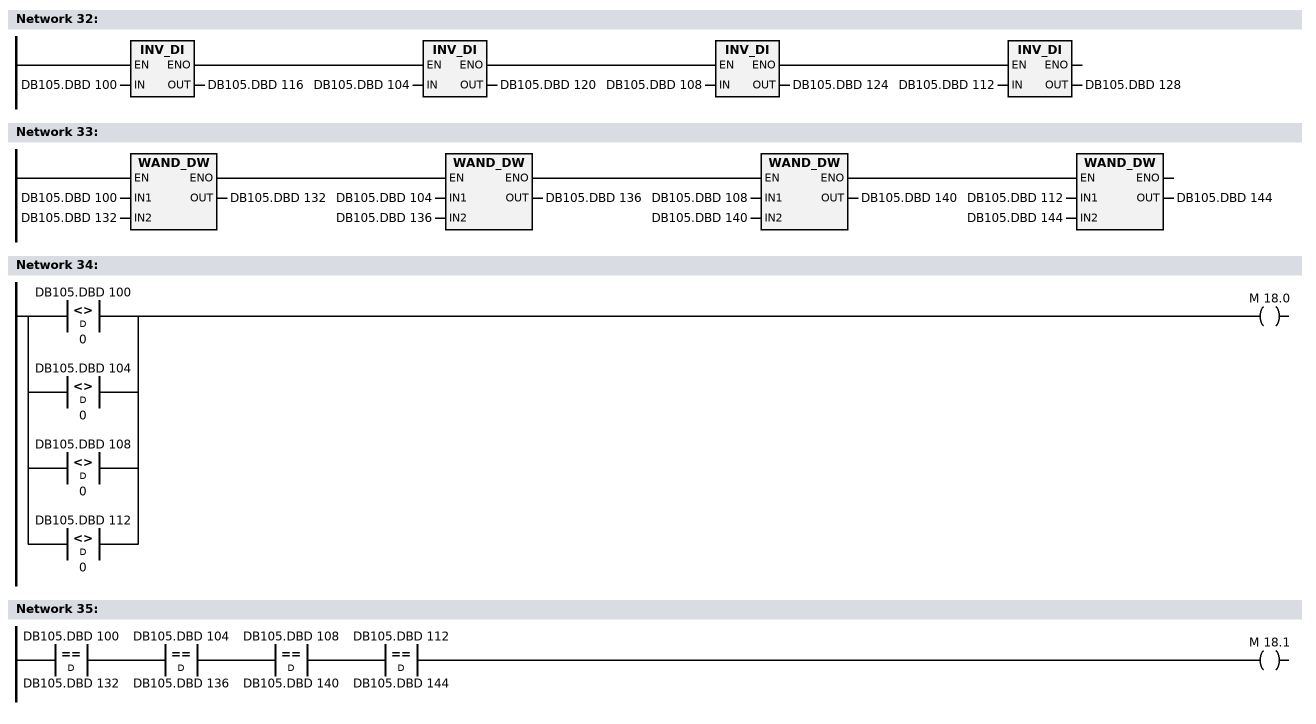
NETWORK
TITLE =
      A(;
      A(;
      A(;
      L     DB105.DBD 100;
      INVD;
      T     DB105.DBD 116;
      SET;
      SAVE;
      CLR;
      A     BR;
      );
      JNB   M001;
      L     DB105.DBD 104;
      INVD;
      T     DB105.DBD 120;
      SET;
      SAVE;
      CLR;
M001: A     BR;
      );
      JNB   M002;
      L     DB105.DBD 108;
      INVD;
      T     DB105.DBD 124;
      SET;
      SAVE;
      CLR;
M002: A     BR;
      );
      JNB   M003;
      L     DB105.DBD 112;
      INVD;
      T     DB105.DBD 128;
M003: NOP   0;
NETWORK
TITLE =
      A(;
      A(;
      A(;
      L     DB105.DBD 100;
      L     DB105.DBD 132;
      AD;
      T     DB105.DBD 132;
      SET;
      SAVE;
      CLR;
      A     BR;
      );
      JNB   M004;
      L     DB105.DBD 104;
      L     DB105.DBD 136;
      AD;
      T     DB105.DBD 136;
      SET;
      SAVE;
      CLR;
M004: A     BR;
      );
      JNB   M005;
      L     DB105.DBD 108;
      L     DB105.DBD 140;
      AD;
      T     DB105.DBD 140;
      SET;
      SAVE;
      CLR;
M005: A     BR;
      );
      JNB   M006;
      L     DB105.DBD 112;
      L     DB105.DBD 144;
      AD;
      T     DB105.DBD 144;
M006: NOP   0;
NETWORK
TITLE =
      O(;
      L     DB105.DBD 100;
      L     0;
      <>D;
      );
      O(;
      L     DB105.DBD 104;
      L     0;
      <>D;
      );
      O(;
      L     DB105.DBD 108;
      L     0;
      <>D;
      );
      O(;
      L     DB105.DBD 112;
      L     0;
      <>D;
      );
      =     M 18.0;
NETWORK
TITLE =
      A(;
      L     DB105.DBD 100;
      L     DB105.DBD 132;
      ==D;
      );
      A(;
      L     DB105.DBD 104;
      L     DB105.DBD 136;
      ==D;
      );
      A(;
      L     DB105.DBD 108;
      L     DB105.DBD 140;
      ==D;
      );
      A(;
      L     DB105.DBD 112;
      L     DB105.DBD 144;
      ==D;
      );
      =     M 18.1;
END_FUNCTION

FUNCTION FC 119 : VOID
VERSION : 0.1
BEGIN
// (block stored without names or comments; labels and parameter names are numbered)
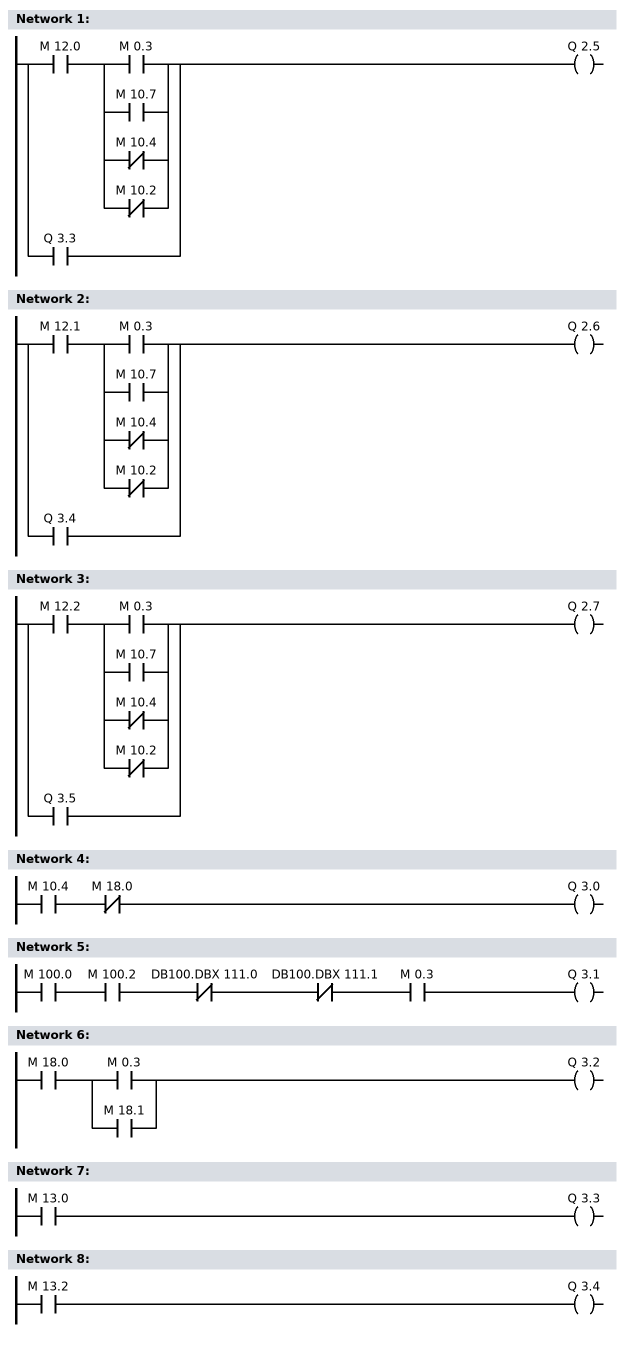
NETWORK
TITLE =
      A     M 12.0;
      A(;
      O     M 0.3;
      O     M 10.7;
      ON    M 10.4;
      ON    M 10.2;
      );
      O     Q 3.3;
      =     Q 2.5;
NETWORK
TITLE =
      A     M 12.1;
      A(;
      O     M 0.3;
      O     M 10.7;
      ON    M 10.4;
      ON    M 10.2;
      );
      O     Q 3.4;
      =     Q 2.6;
NETWORK
TITLE =
      A     M 12.2;
      A(;
      O     M 0.3;
      O     M 10.7;
      ON    M 10.4;
      ON    M 10.2;
      );
      O     Q 3.5;
      =     Q 2.7;
NETWORK
TITLE =
      A     M 10.4;
      AN    M 18.0;
      =     Q 3.0;
NETWORK
TITLE =
      A     M 100.0;
      A     M 100.2;
      AN    DB100.DBX 111.0;
      AN    DB100.DBX 111.1;
      A     M 0.3;
      =     Q 3.1;
NETWORK
TITLE =
      A     M 18.0;
      A(;
      O     M 0.3;
      O     M 18.1;
      );
      =     Q 3.2;
NETWORK
TITLE =
      A     M 13.0;
      =     Q 3.3;
NETWORK
TITLE =
      A     M 13.2;
      =     Q 3.4;
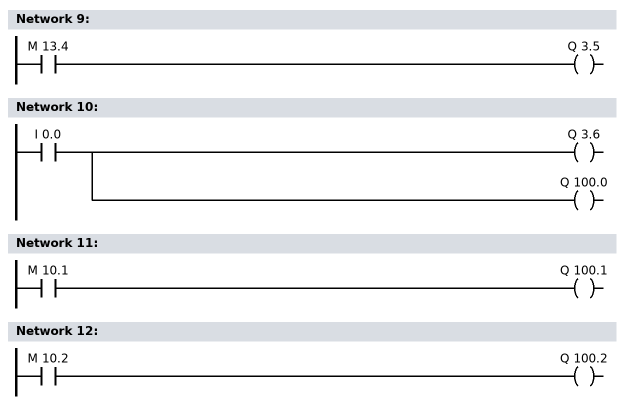
NETWORK
TITLE =
      A     M 13.4;
      =     Q 3.5;
NETWORK
TITLE =
      A     I 0.0;
      =     Q 3.6;
      =     Q 100.0;
NETWORK
TITLE =
      A     M 10.1;
      =     Q 100.1;
NETWORK
TITLE =
      A     M 10.2;
      =     Q 100.2;
END_FUNCTION

FUNCTION FC 140 : VOID
VERSION : 0.1
BEGIN
// (block stored without names or comments; labels and parameter names are numbered)
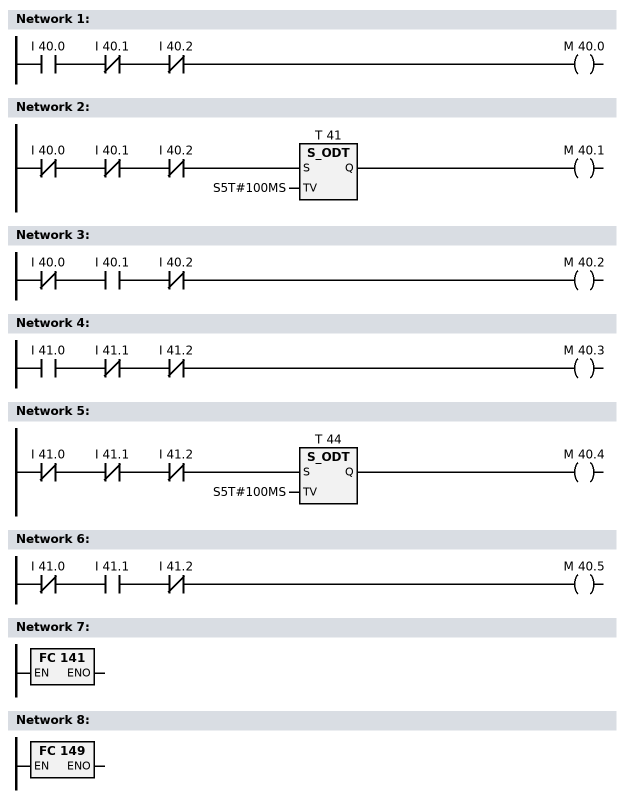
NETWORK
TITLE =
      A     I 40.0;
      AN    I 40.1;
      AN    I 40.2;
      =     M 40.0;
NETWORK
TITLE =
      AN    I 40.0;
      AN    I 40.1;
      AN    I 40.2;
      L     S5T#100MS;
      SD    T 41;
      NOP   0;
      NOP   0;
      NOP   0;
      A     T 41;
      =     M 40.1;
NETWORK
TITLE =
      AN    I 40.0;
      A     I 40.1;
      AN    I 40.2;
      =     M 40.2;
NETWORK
TITLE =
      A     I 41.0;
      AN    I 41.1;
      AN    I 41.2;
      =     M 40.3;
NETWORK
TITLE =
      AN    I 41.0;
      AN    I 41.1;
      AN    I 41.2;
      L     S5T#100MS;
      SD    T 44;
      NOP   0;
      NOP   0;
      NOP   0;
      A     T 44;
      =     M 40.4;
NETWORK
TITLE =
      AN    I 41.0;
      A     I 41.1;
      AN    I 41.2;
      =     M 40.5;
NETWORK
TITLE =
      CALL  FC 141;
      NOP   0;
NETWORK
TITLE =
      CALL  FC 149;
      NOP   0;
END_FUNCTION

FUNCTION FC 141 : VOID
VERSION : 0.1
BEGIN
// (block stored without names or comments; labels and parameter names are numbered)
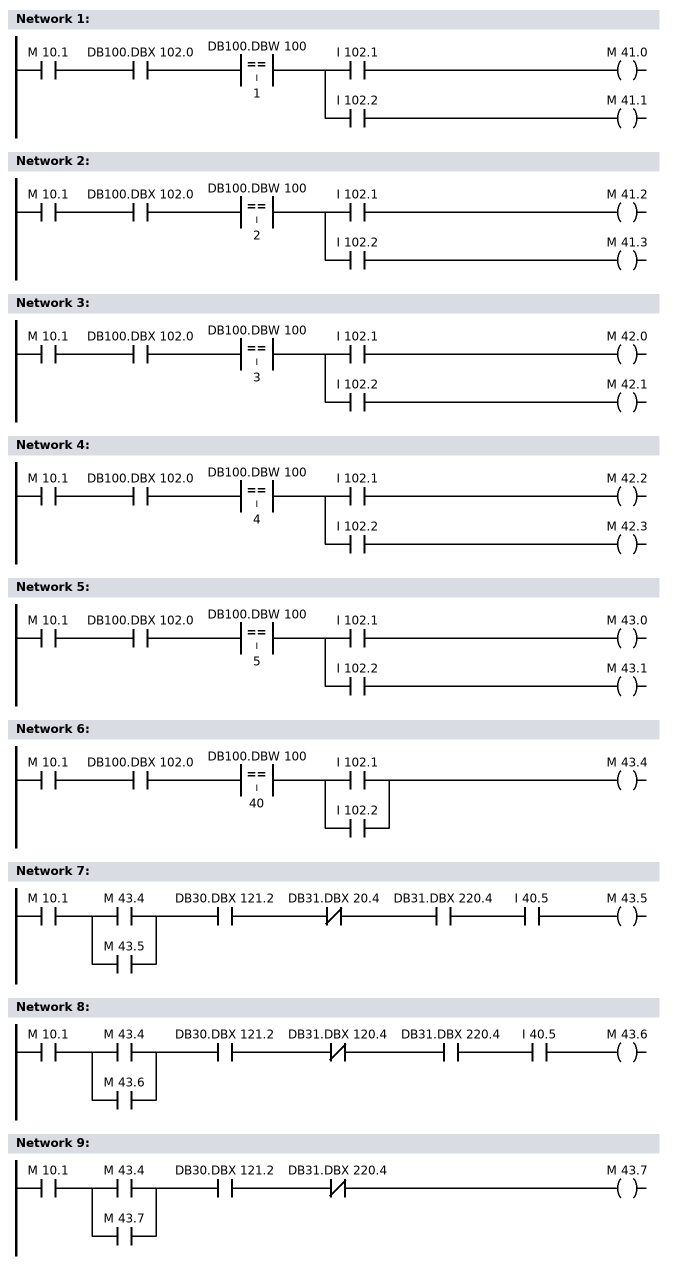
NETWORK
TITLE =
      A     M 10.1;
      A     DB100.DBX 102.0;
      A(;
      L     DB100.DBW 100;
      L     1;
      ==I;
      );
      =     L 0.0;
      A     L 0.0;
      A     I 102.1;
      =     M 41.0;
      A     L 0.0;
      A     I 102.2;
      =     M 41.1;
NETWORK
TITLE =
      A     M 10.1;
      A     DB100.DBX 102.0;
      A(;
      L     DB100.DBW 100;
      L     2;
      ==I;
      );
      =     L 0.0;
      A     L 0.0;
      A     I 102.1;
      =     M 41.2;
      A     L 0.0;
      A     I 102.2;
      =     M 41.3;
NETWORK
TITLE =
      A     M 10.1;
      A     DB100.DBX 102.0;
      A(;
      L     DB100.DBW 100;
      L     3;
      ==I;
      );
      =     L 0.0;
      A     L 0.0;
      A     I 102.1;
      =     M 42.0;
      A     L 0.0;
      A     I 102.2;
      =     M 42.1;
NETWORK
TITLE =
      A     M 10.1;
      A     DB100.DBX 102.0;
      A(;
      L     DB100.DBW 100;
      L     4;
      ==I;
      );
      =     L 0.0;
      A     L 0.0;
      A     I 102.1;
      =     M 42.2;
      A     L 0.0;
      A     I 102.2;
      =     M 42.3;
NETWORK
TITLE =
      A     M 10.1;
      A     DB100.DBX 102.0;
      A(;
      L     DB100.DBW 100;
      L     5;
      ==I;
      );
      =     L 0.0;
      A     L 0.0;
      A     I 102.1;
      =     M 43.0;
      A     L 0.0;
      A     I 102.2;
      =     M 43.1;
NETWORK
TITLE =
      A     M 10.1;
      A     DB100.DBX 102.0;
      A(;
      L     DB100.DBW 100;
      L     40;
      ==I;
      );
      A(;
      O     I 102.1;
      O     I 102.2;
      );
      =     M 43.4;
NETWORK
TITLE =
      A     M 10.1;
      A(;
      O     M 43.4;
      O     M 43.5;
      );
      A     DB30.DBX 121.2;
      AN    DB31.DBX 20.4;
      A     DB31.DBX 220.4;
      A     I 40.5;
      =     M 43.5;
NETWORK
TITLE =
      A     M 10.1;
      A(;
      O     M 43.4;
      O     M 43.6;
      );
      A     DB30.DBX 121.2;
      AN    DB31.DBX 120.4;
      A     DB31.DBX 220.4;
      A     I 40.5;
      =     M 43.6;
NETWORK
TITLE =
      A     M 10.1;
      A(;
      O     M 43.4;
      O     M 43.7;
      );
      A     DB30.DBX 121.2;
      AN    DB31.DBX 220.4;
      =     M 43.7;
END_FUNCTION

FUNCTION FC 142 : VOID
VERSION : 0.1
BEGIN
// (block stored without names or comments; labels and parameter names are numbered)
END_FUNCTION

FUNCTION FC 149 : VOID
VERSION : 0.1
BEGIN
// (block stored without names or comments; labels and parameter names are numbered)
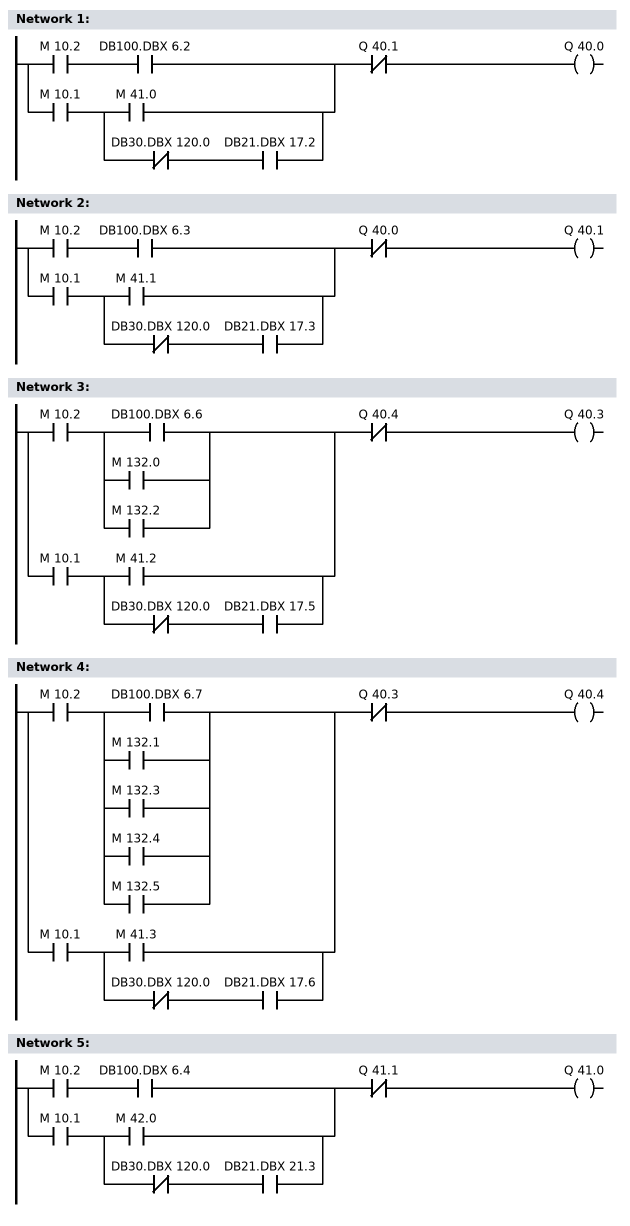
NETWORK
TITLE =
      A(;
      A     M 10.2;
      A     DB100.DBX 6.2;
      O;
      A     M 10.1;
      A(;
      O     M 41.0;
      O;
      AN    DB30.DBX 120.0;
      A     DB21.DBX 17.2;
      );
      );
      AN    Q 40.1;
      =     Q 40.0;
NETWORK
TITLE =
      A(;
      A     M 10.2;
      A     DB100.DBX 6.3;
      O;
      A     M 10.1;
      A(;
      O     M 41.1;
      O;
      AN    DB30.DBX 120.0;
      A     DB21.DBX 17.3;
      );
      );
      AN    Q 40.0;
      =     Q 40.1;
NETWORK
TITLE =
      A(;
      A     M 10.2;
      A(;
      O     DB100.DBX 6.6;
      O     M 132.0;
      O     M 132.2;
      );
      O;
      A     M 10.1;
      A(;
      O     M 41.2;
      O;
      AN    DB30.DBX 120.0;
      A     DB21.DBX 17.5;
      );
      );
      AN    Q 40.4;
      =     Q 40.3;
NETWORK
TITLE =
      A(;
      A     M 10.2;
      A(;
      O     DB100.DBX 6.7;
      O     M 132.1;
      O     M 132.3;
      O     M 132.4;
      O     M 132.5;
      );
      O;
      A     M 10.1;
      A(;
      O     M 41.3;
      O;
      AN    DB30.DBX 120.0;
      A     DB21.DBX 17.6;
      );
      );
      AN    Q 40.3;
      =     Q 40.4;
NETWORK
TITLE =
      A(;
      A     M 10.2;
      A     DB100.DBX 6.4;
      O;
      A     M 10.1;
      A(;
      O     M 42.0;
      O;
      AN    DB30.DBX 120.0;
      A     DB21.DBX 21.3;
      );
      );
      AN    Q 41.1;
      =     Q 41.0;
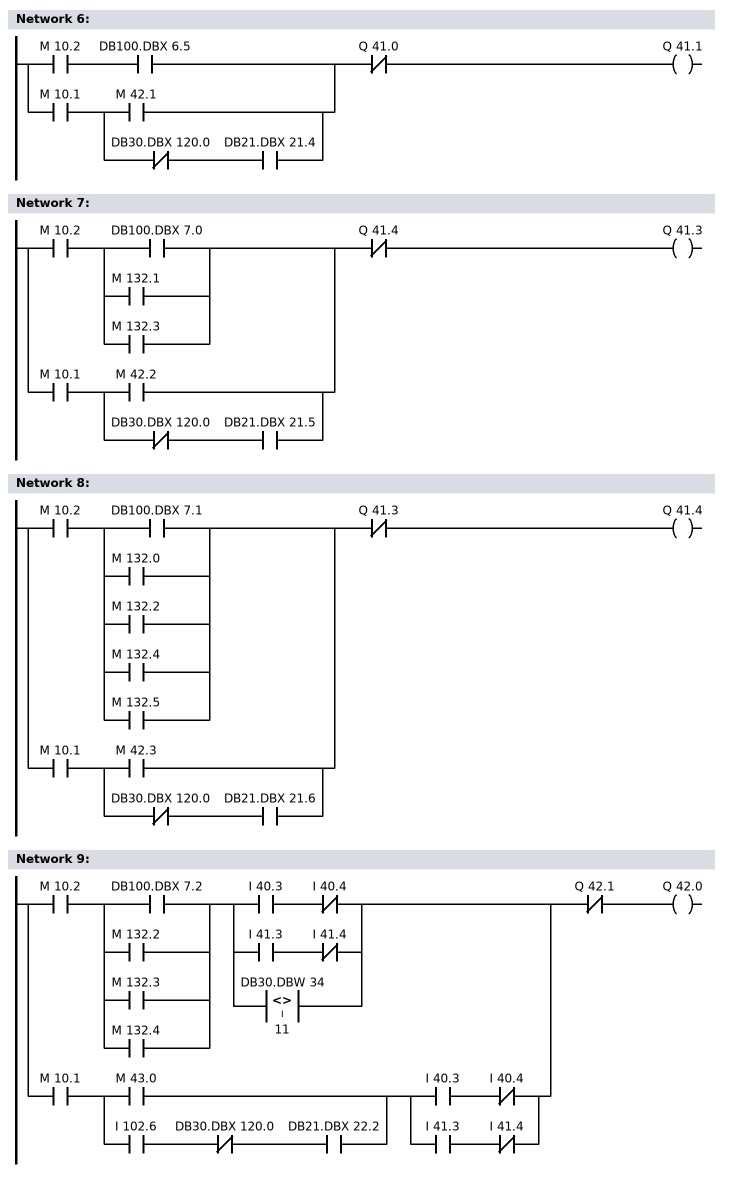
NETWORK
TITLE =
      A(;
      A     M 10.2;
      A     DB100.DBX 6.5;
      O;
      A     M 10.1;
      A(;
      O     M 42.1;
      O;
      AN    DB30.DBX 120.0;
      A     DB21.DBX 21.4;
      );
      );
      AN    Q 41.0;
      =     Q 41.1;
NETWORK
TITLE =
      A(;
      A     M 10.2;
      A(;
      O     DB100.DBX 7.0;
      O     M 132.1;
      O     M 132.3;
      );
      O;
      A     M 10.1;
      A(;
      O     M 42.2;
      O;
      AN    DB30.DBX 120.0;
      A     DB21.DBX 21.5;
      );
      );
      AN    Q 41.4;
      =     Q 41.3;
NETWORK
TITLE =
      A(;
      A     M 10.2;
      A(;
      O     DB100.DBX 7.1;
      O     M 132.0;
      O     M 132.2;
      O     M 132.4;
      O     M 132.5;
      );
      O;
      A     M 10.1;
      A(;
      O     M 42.3;
      O;
      AN    DB30.DBX 120.0;
      A     DB21.DBX 21.6;
      );
      );
      AN    Q 41.3;
      =     Q 41.4;
NETWORK
TITLE =
      A(;
      A     M 10.2;
      A(;
      O     DB100.DBX 7.2;
      O     M 132.2;
      O     M 132.3;
      O     M 132.4;
      );
      A(;
      A     I 40.3;
      AN    I 40.4;
      O;
      A     I 41.3;
      AN    I 41.4;
      O(;
      L     DB30.DBW 34;
      L     11;
      <>I;
      );
      );
      O;
      A     M 10.1;
      A(;
      O     M 43.0;
      O;
      A     I 102.6;
      AN    DB30.DBX 120.0;
      A     DB21.DBX 22.2;
      );
      A(;
      A     I 40.3;
      AN    I 40.4;
      O;
      A     I 41.3;
      AN    I 41.4;
      );
      );
      AN    Q 42.1;
      =     Q 42.0;
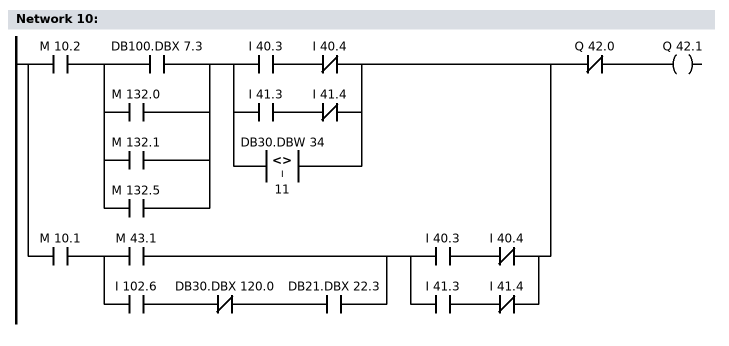
NETWORK
TITLE =
      A(;
      A     M 10.2;
      A(;
      O     DB100.DBX 7.3;
      O     M 132.0;
      O     M 132.1;
      O     M 132.5;
      );
      A(;
      A     I 40.3;
      AN    I 40.4;
      O;
      A     I 41.3;
      AN    I 41.4;
      O(;
      L     DB30.DBW 34;
      L     11;
      <>I;
      );
      );
      O;
      A     M 10.1;
      A(;
      O     M 43.1;
      O;
      A     I 102.6;
      AN    DB30.DBX 120.0;
      A     DB21.DBX 22.3;
      );
      A(;
      A     I 40.3;
      AN    I 40.4;
      O;
      A     I 41.3;
      AN    I 41.4;
      );
      );
      AN    Q 42.0;
      =     Q 42.1;
NETWORK
TITLE =
END_FUNCTION

FUNCTION FC 160 : VOID
VERSION : 0.1
BEGIN
// (block stored without names or comments; labels and parameter names are numbered)
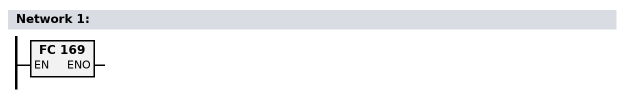
NETWORK
TITLE =
      CALL  FC 169;
      NOP   0;
END_FUNCTION

FUNCTION FC 169 : VOID
VERSION : 0.1
BEGIN
// (block stored without names or comments; labels and parameter names are numbered)
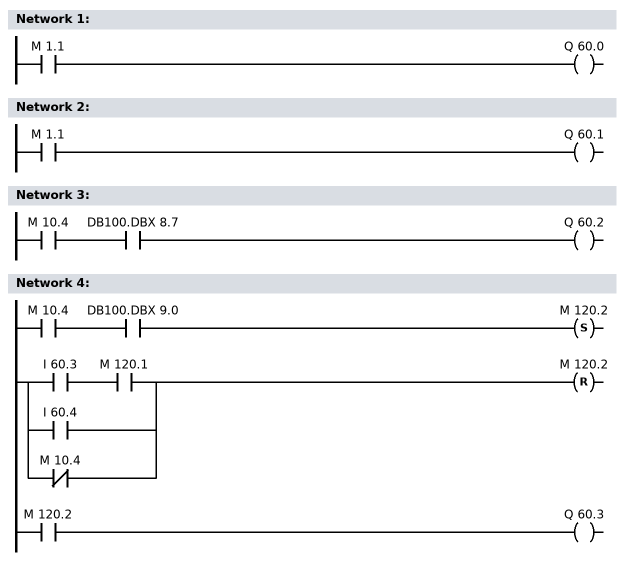
NETWORK
TITLE =
      A     M 1.1;
      =     Q 60.0;
NETWORK
TITLE =
      A     M 1.1;
      =     Q 60.1;
NETWORK
TITLE =
      A     M 10.4;
      A     DB100.DBX 8.7;
      =     Q 60.2;
NETWORK
TITLE =
      A     M 10.4;
      A     DB100.DBX 9.0;
      S     M 120.2;
      A(;
      A     I 60.3;
      A     M 120.1;
      O     I 60.4;
      ON    M 10.4;
      );
      R     M 120.2;
      A     M 120.2;
      =     Q 60.3;
NETWORK
TITLE =
      A(;
      A     M 10.4;
      A     M 120.2;
      A     DB100.DBX 10.0;
      S     M 120.1;
      A(;
      A     M 120.1;
      A     I 60.4;
      ON    M 10.4;
      );
      R     M 120.1;
      A     M 120.1;
      );
      A     I 60.3;
      S     M 120.3;
      A(;
      A     M 120.3;
      A     I 60.4;
      ON    M 10.4;
      );
      R     M 120.3;
      A     M 120.3;
      =     Q 60.5;
      =     Q 60.6;
END_FUNCTION

FUNCTION FC 170 : VOID
VERSION : 0.1
BEGIN
// (block stored without names or comments; labels and parameter names are numbered)
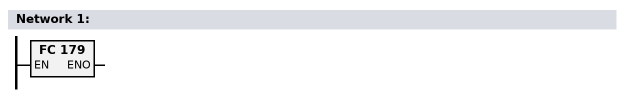
NETWORK
TITLE =
      CALL  FC 179;
      NOP   0;
END_FUNCTION

FUNCTION FC 179 : VOID
VERSION : 0.1
BEGIN
// (block stored without names or comments; labels and parameter names are numbered)
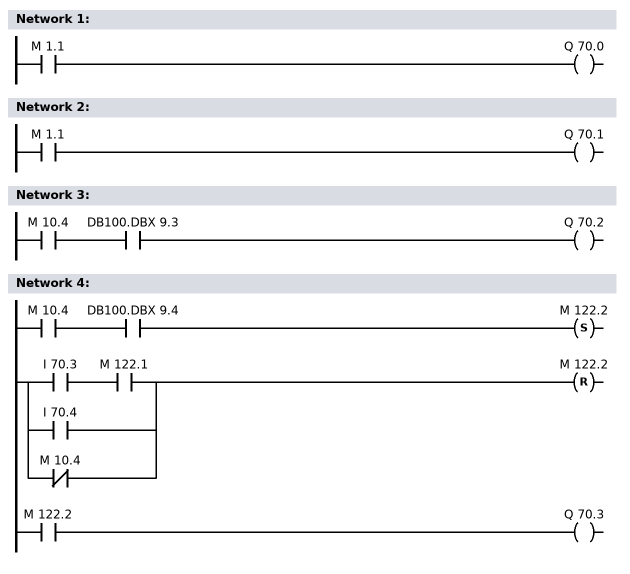
NETWORK
TITLE =
      A     M 1.1;
      =     Q 70.0;
NETWORK
TITLE =
      A     M 1.1;
      =     Q 70.1;
NETWORK
TITLE =
      A     M 10.4;
      A     DB100.DBX 9.3;
      =     Q 70.2;
NETWORK
TITLE =
      A     M 10.4;
      A     DB100.DBX 9.4;
      S     M 122.2;
      A(;
      A     I 70.3;
      A     M 122.1;
      O     I 70.4;
      ON    M 10.4;
      );
      R     M 122.2;
      A     M 122.2;
      =     Q 70.3;
NETWORK
TITLE =
      A(;
      A     M 10.4;
      A     M 122.2;
      A     DB100.DBX 10.1;
      S     M 122.1;
      A(;
      A     M 122.1;
      A     I 70.4;
      ON    M 10.4;
      );
      R     M 122.1;
      A     M 122.1;
      );
      A     I 70.3;
      S     M 122.3;
      A(;
      A     M 122.3;
      A     I 70.4;
      ON    M 10.4;
      );
      R     M 122.3;
      A     M 122.3;
      =     Q 70.5;
      =     Q 70.6;
END_FUNCTION

FUNCTION FC 180 : VOID
VERSION : 0.1
BEGIN
// (block stored without names or comments; labels and parameter names are numbered)
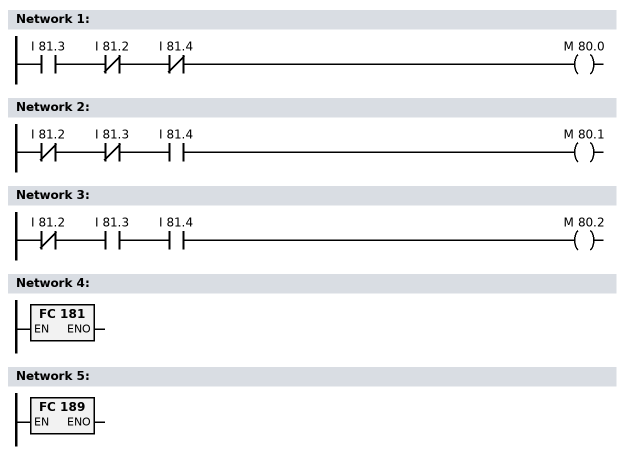
NETWORK
TITLE =
      A     I 81.3;
      AN    I 81.2;
      AN    I 81.4;
      =     M 80.0;
NETWORK
TITLE =
      AN    I 81.2;
      AN    I 81.3;
      A     I 81.4;
      =     M 80.1;
NETWORK
TITLE =
      AN    I 81.2;
      A     I 81.3;
      A     I 81.4;
      =     M 80.2;
NETWORK
TITLE =
      CALL  FC 181;
      NOP   0;
NETWORK
TITLE =
      CALL  FC 189;
      NOP   0;
END_FUNCTION

FUNCTION FC 181 : VOID
VERSION : 0.1
BEGIN
// (block stored without names or comments; labels and parameter names are numbered)
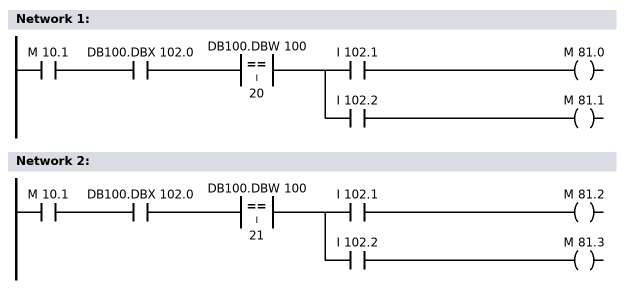
NETWORK
TITLE =
      A     M 10.1;
      A     DB100.DBX 102.0;
      A(;
      L     DB100.DBW 100;
      L     20;
      ==I;
      );
      =     L 0.0;
      A     L 0.0;
      A     I 102.1;
      =     M 81.0;
      A     L 0.0;
      A     I 102.2;
      =     M 81.1;
NETWORK
TITLE =
      A     M 10.1;
      A     DB100.DBX 102.0;
      A(;
      L     DB100.DBW 100;
      L     21;
      ==I;
      );
      =     L 0.0;
      A     L 0.0;
      A     I 102.1;
      =     M 81.2;
      A     L 0.0;
      A     I 102.2;
      =     M 81.3;
END_FUNCTION

FUNCTION FC 182 : VOID
VERSION : 0.1
BEGIN
// (block stored without names or comments; labels and parameter names are numbered)
END_FUNCTION

FUNCTION FC 189 : VOID
VERSION : 0.1
BEGIN
// (block stored without names or comments; labels and parameter names are numbered)
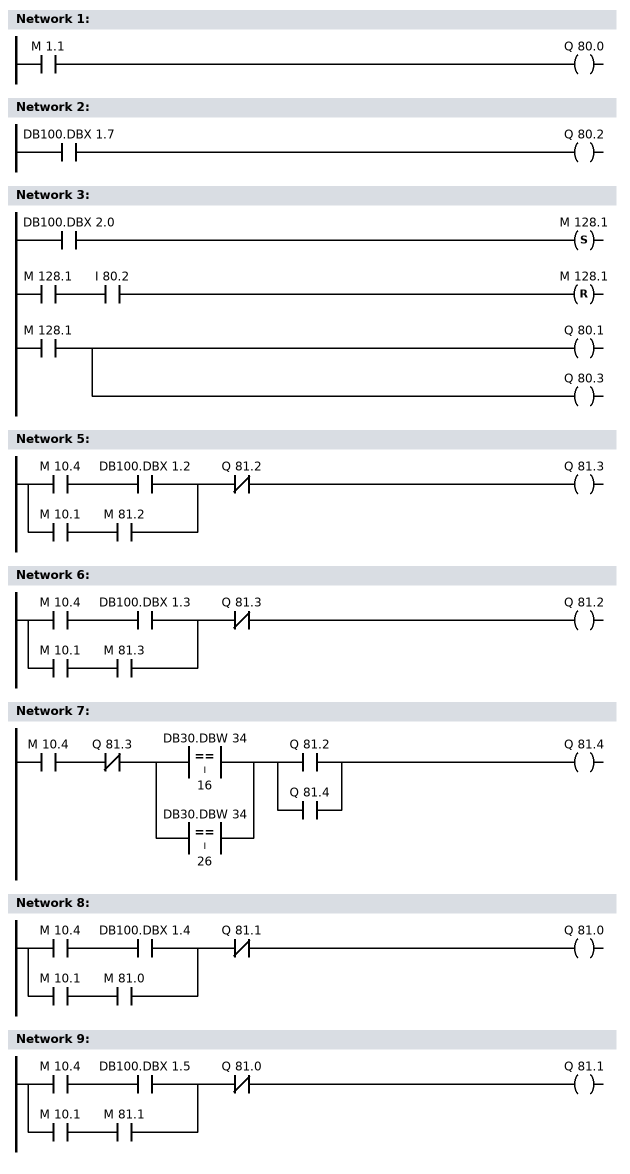
NETWORK
TITLE =
      A     M 1.1;
      =     Q 80.0;
NETWORK
TITLE =
      A     DB100.DBX 1.7;
      =     Q 80.2;
NETWORK
TITLE =
      A     DB100.DBX 2.0;
      S     M 128.1;
      A     M 128.1;
      A     I 80.2;
      R     M 128.1;
      A     M 128.1;
      =     Q 80.1;
      =     Q 80.3;
NETWORK
TITLE =
NETWORK
TITLE =
      A(;
      A     M 10.4;
      A     DB100.DBX 1.2;
      O;
      A     M 10.1;
      A     M 81.2;
      );
      AN    Q 81.2;
      =     Q 81.3;
NETWORK
TITLE =
      A(;
      A     M 10.4;
      A     DB100.DBX 1.3;
      O;
      A     M 10.1;
      A     M 81.3;
      );
      AN    Q 81.3;
      =     Q 81.2;
NETWORK
TITLE =
      A     M 10.4;
      AN    Q 81.3;
      A(;
      O(;
      L     DB30.DBW 34;
      L     16;
      ==I;
      );
      O(;
      L     DB30.DBW 34;
      L     26;
      ==I;
      );
      );
      A(;
      O     Q 81.2;
      O     Q 81.4;
      );
      =     Q 81.4;
NETWORK
TITLE =
      A(;
      A     M 10.4;
      A     DB100.DBX 1.4;
      O;
      A     M 10.1;
      A     M 81.0;
      );
      AN    Q 81.1;
      =     Q 81.0;
NETWORK
TITLE =
      A(;
      A     M 10.4;
      A     DB100.DBX 1.5;
      O;
      A     M 10.1;
      A     M 81.1;
      );
      AN    Q 81.0;
      =     Q 81.1;
END_FUNCTION

FUNCTION FC 190 : VOID
VERSION : 0.1
BEGIN
// (block stored without names or comments; labels and parameter names are numbered)
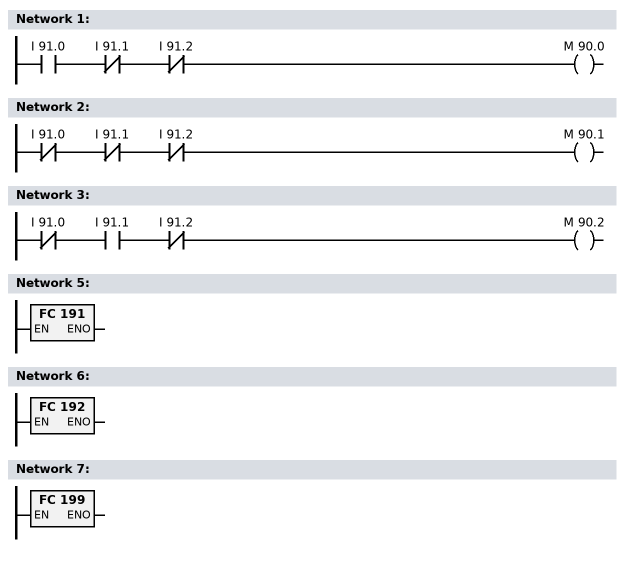
NETWORK
TITLE =
      A     I 91.0;
      AN    I 91.1;
      AN    I 91.2;
      =     M 90.0;
NETWORK
TITLE =
      AN    I 91.0;
      AN    I 91.1;
      AN    I 91.2;
      =     M 90.1;
NETWORK
TITLE =
      AN    I 91.0;
      A     I 91.1;
      AN    I 91.2;
      =     M 90.2;
NETWORK
TITLE =
NETWORK
TITLE =
      CALL  FC 191;
      NOP   0;
NETWORK
TITLE =
      CALL  FC 192;
      NOP   0;
NETWORK
TITLE =
      CALL  FC 199;
      NOP   0;
END_FUNCTION

FUNCTION FC 191 : VOID
VERSION : 0.1
BEGIN
// (block stored without names or comments; labels and parameter names are numbered)
NETWORK
TITLE =
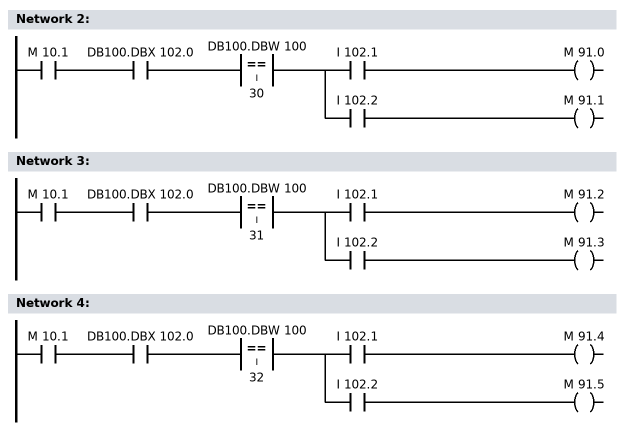
NETWORK
TITLE =
      A     M 10.1;
      A     DB100.DBX 102.0;
      A(;
      L     DB100.DBW 100;
      L     30;
      ==I;
      );
      =     L 0.0;
      A     L 0.0;
      A     I 102.1;
      =     M 91.0;
      A     L 0.0;
      A     I 102.2;
      =     M 91.1;
NETWORK
TITLE =
      A     M 10.1;
      A     DB100.DBX 102.0;
      A(;
      L     DB100.DBW 100;
      L     31;
      ==I;
      );
      =     L 0.0;
      A     L 0.0;
      A     I 102.1;
      =     M 91.2;
      A     L 0.0;
      A     I 102.2;
      =     M 91.3;
NETWORK
TITLE =
      A     M 10.1;
      A     DB100.DBX 102.0;
      A(;
      L     DB100.DBW 100;
      L     32;
      ==I;
      );
      =     L 0.0;
      A     L 0.0;
      A     I 102.1;
      =     M 91.4;
      A     L 0.0;
      A     I 102.2;
      =     M 91.5;
END_FUNCTION

FUNCTION FC 192 : VOID
VERSION : 0.1
BEGIN
// (block stored without names or comments; labels and parameter names are numbered)
NETWORK
TITLE =
      A(;
      A     M 10.4;
      A     I 90.1;
      A     I 90.3;
      A(;
      ON    M 10.6;
      O     DB100.DBX 4.1;
      );
      AN    M 94.0;
      A     M 90.0;
      S     M 92.0;
      A(;
      A     M 92.0;
      A     M 92.1;
      ON    M 10.4;
      );
      R     M 92.0;
      A     M 92.0;
      );
      S     M 94.0;
      A(;
      A     M 94.0;
      A     I 90.2;
      ON    M 10.4;
      );
      R     M 94.0;
      NOP   0;
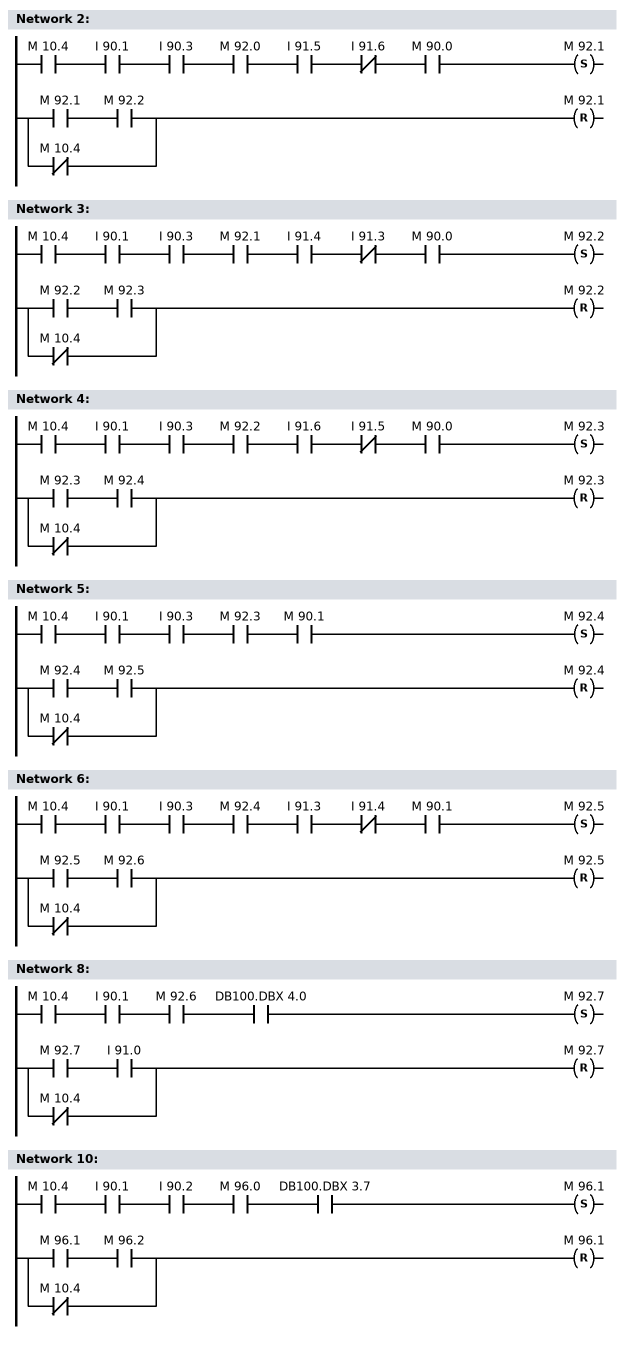
NETWORK
TITLE =
      A     M 10.4;
      A     I 90.1;
      A     I 90.3;
      A     M 92.0;
      A     I 91.5;
      AN    I 91.6;
      A     M 90.0;
      S     M 92.1;
      A(;
      A     M 92.1;
      A     M 92.2;
      ON    M 10.4;
      );
      R     M 92.1;
      NOP   0;
NETWORK
TITLE =
      A     M 10.4;
      A     I 90.1;
      A     I 90.3;
      A     M 92.1;
      A     I 91.4;
      AN    I 91.3;
      A     M 90.0;
      S     M 92.2;
      A(;
      A     M 92.2;
      A     M 92.3;
      ON    M 10.4;
      );
      R     M 92.2;
      NOP   0;
NETWORK
TITLE =
      A     M 10.4;
      A     I 90.1;
      A     I 90.3;
      A     M 92.2;
      A     I 91.6;
      AN    I 91.5;
      A     M 90.0;
      S     M 92.3;
      A(;
      A     M 92.3;
      A     M 92.4;
      ON    M 10.4;
      );
      R     M 92.3;
      NOP   0;
NETWORK
TITLE =
      A     M 10.4;
      A     I 90.1;
      A     I 90.3;
      A     M 92.3;
      A     M 90.1;
      S     M 92.4;
      A(;
      A     M 92.4;
      A     M 92.5;
      ON    M 10.4;
      );
      R     M 92.4;
      NOP   0;
NETWORK
TITLE =
      A     M 10.4;
      A     I 90.1;
      A     I 90.3;
      A     M 92.4;
      A     I 91.3;
      AN    I 91.4;
      A     M 90.1;
      S     M 92.5;
      A(;
      A     M 92.5;
      A     M 92.6;
      ON    M 10.4;
      );
      R     M 92.5;
      NOP   0;
NETWORK
TITLE =
      A(;
      A     M 10.4;
      A     I 90.1;
      A(;
      A     I 90.3;
      A     M 92.5;
      ON    M 94.6;
      );
      A     I 91.5;
      AN    I 91.6;
      A     I 91.3;
      AN    I 91.4;
      A     M 90.1;
      S     M 92.6;
      A(;
      A     M 92.6;
      A     M 92.7;
      ON    M 10.4;
      );
      R     M 92.6;
      A     M 92.6;
      );
      S     M 94.6;
      A     M 94.6;
      AN    M 10.4;
      R     M 94.6;
      NOP   0;
NETWORK
TITLE =
      A     M 10.4;
      A     I 90.1;
      A     M 92.6;
      A     DB100.DBX 4.0;
      S     M 92.7;
      A(;
      A     M 92.7;
      A     I 91.0;
      ON    M 10.4;
      );
      R     M 92.7;
      NOP   0;
NETWORK
TITLE =
      A(;
      A     M 10.4;
      A     I 90.1;
      A     I 90.2;
      AN    M 96.7;
      AN    M 98.0;
      A     M 90.0;
      S     M 96.0;
      A(;
      A     M 96.0;
      A     M 96.1;
      ON    M 10.4;
      );
      R     M 96.0;
      A     M 96.0;
      );
      S     M 98.0;
      A(;
      A     M 98.0;
      A     I 90.3;
      ON    M 10.4;
      );
      R     M 98.0;
      NOP   0;
NETWORK
TITLE =
      A     M 10.4;
      A     I 90.1;
      A     I 90.2;
      A     M 96.0;
      A     DB100.DBX 3.7;
      S     M 96.1;
      A(;
      A     M 96.1;
      A     M 96.2;
      ON    M 10.4;
      );
      R     M 96.1;
      NOP   0;
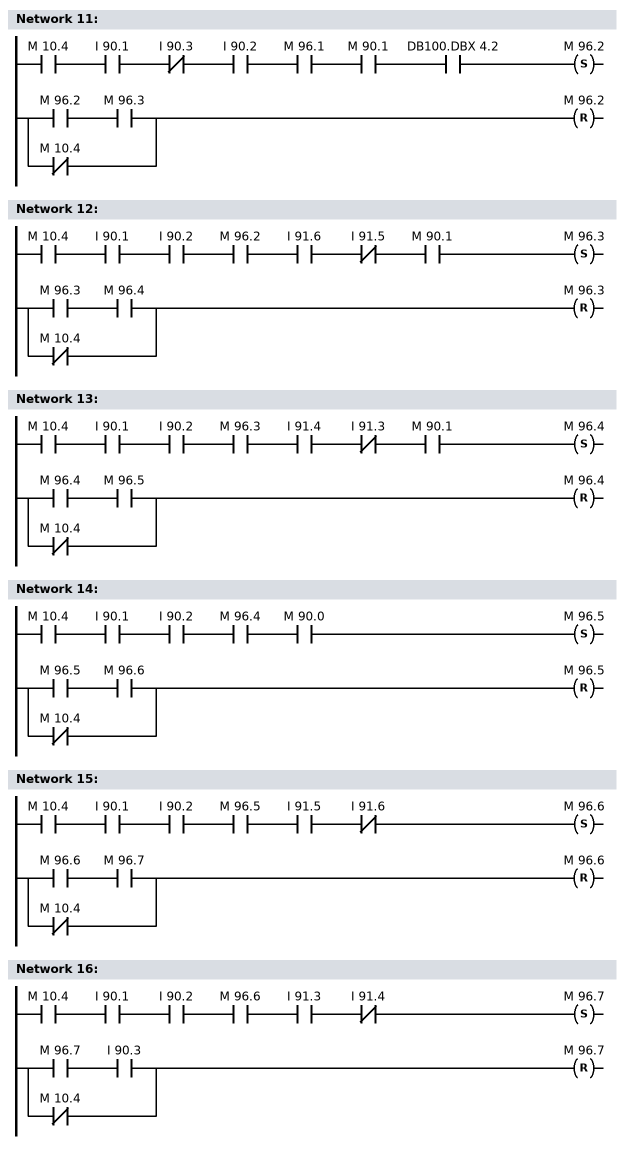
NETWORK
TITLE =
      A     M 10.4;
      A     I 90.1;
      AN    I 90.3;
      A     I 90.2;
      A     M 96.1;
      A     M 90.1;
      A     DB100.DBX 4.2;
      S     M 96.2;
      A(;
      A     M 96.2;
      A     M 96.3;
      ON    M 10.4;
      );
      R     M 96.2;
      NOP   0;
NETWORK
TITLE =
      A     M 10.4;
      A     I 90.1;
      A     I 90.2;
      A     M 96.2;
      A     I 91.6;
      AN    I 91.5;
      A     M 90.1;
      S     M 96.3;
      A(;
      A     M 96.3;
      A     M 96.4;
      ON    M 10.4;
      );
      R     M 96.3;
      NOP   0;
NETWORK
TITLE =
      A     M 10.4;
      A     I 90.1;
      A     I 90.2;
      A     M 96.3;
      A     I 91.4;
      AN    I 91.3;
      A     M 90.1;
      S     M 96.4;
      A(;
      A     M 96.4;
      A     M 96.5;
      ON    M 10.4;
      );
      R     M 96.4;
      NOP   0;
NETWORK
TITLE =
      A     M 10.4;
      A     I 90.1;
      A     I 90.2;
      A     M 96.4;
      A     M 90.0;
      S     M 96.5;
      A(;
      A     M 96.5;
      A     M 96.6;
      ON    M 10.4;
      );
      R     M 96.5;
      NOP   0;
NETWORK
TITLE =
      A     M 10.4;
      A     I 90.1;
      A     I 90.2;
      A     M 96.5;
      A     I 91.5;
      AN    I 91.6;
      S     M 96.6;
      A(;
      A     M 96.6;
      A     M 96.7;
      ON    M 10.4;
      );
      R     M 96.6;
      NOP   0;
NETWORK
TITLE =
      A     M 10.4;
      A     I 90.1;
      A     I 90.2;
      A     M 96.6;
      A     I 91.3;
      AN    I 91.4;
      S     M 96.7;
      A(;
      A     M 96.7;
      A     I 90.3;
      ON    M 10.4;
      );
      R     M 96.7;
      NOP   0;
END_FUNCTION

FUNCTION FC 199 : VOID
VERSION : 0.1
BEGIN
// (block stored without names or comments; labels and parameter names are numbered)
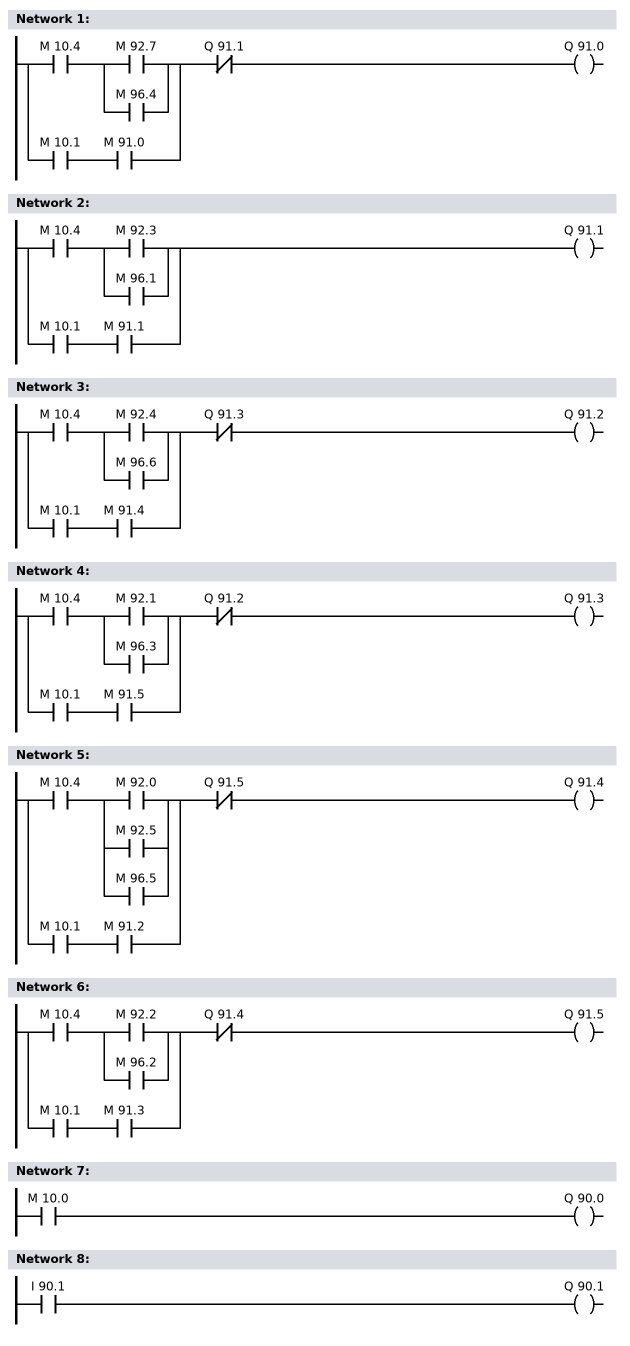
NETWORK
TITLE =
      A(;
      A     M 10.4;
      A(;
      O     M 92.7;
      O     M 96.4;
      );
      O;
      A     M 10.1;
      A     M 91.0;
      );
      AN    Q 91.1;
      =     Q 91.0;
NETWORK
TITLE =
      A     M 10.4;
      A(;
      O     M 92.3;
      O     M 96.1;
      );
      O;
      A     M 10.1;
      A     M 91.1;
      =     Q 91.1;
NETWORK
TITLE =
      A(;
      A     M 10.4;
      A(;
      O     M 92.4;
      O     M 96.6;
      );
      O;
      A     M 10.1;
      A     M 91.4;
      );
      AN    Q 91.3;
      =     Q 91.2;
NETWORK
TITLE =
      A(;
      A     M 10.4;
      A(;
      O     M 92.1;
      O     M 96.3;
      );
      O;
      A     M 10.1;
      A     M 91.5;
      );
      AN    Q 91.2;
      =     Q 91.3;
NETWORK
TITLE =
      A(;
      A     M 10.4;
      A(;
      O     M 92.0;
      O     M 92.5;
      O     M 96.5;
      );
      O;
      A     M 10.1;
      A     M 91.2;
      );
      AN    Q 91.5;
      =     Q 91.4;
NETWORK
TITLE =
      A(;
      A     M 10.4;
      A(;
      O     M 92.2;
      O     M 96.2;
      );
      O;
      A     M 10.1;
      A     M 91.3;
      );
      AN    Q 91.4;
      =     Q 91.5;
NETWORK
TITLE =
      A     M 10.0;
      =     Q 90.0;
NETWORK
TITLE =
      A     I 90.1;
      =     Q 90.1;
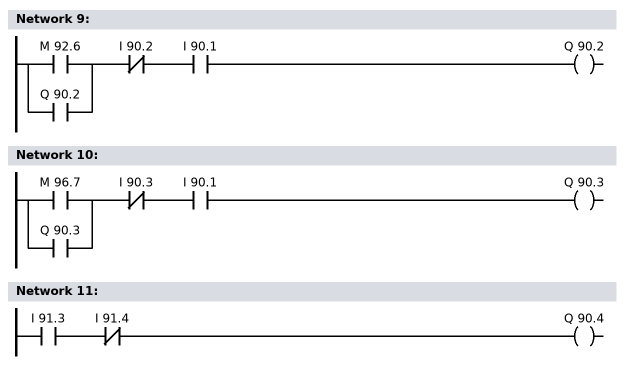
NETWORK
TITLE =
      A(;
      O     M 92.6;
      O     Q 90.2;
      );
      AN    I 90.2;
      A     I 90.1;
      =     Q 90.2;
NETWORK
TITLE =
      A(;
      O     M 96.7;
      O     Q 90.3;
      );
      AN    I 90.3;
      A     I 90.1;
      =     Q 90.3;
NETWORK
TITLE =
      A     I 91.3;
      AN    I 91.4;
      =     Q 90.4;
END_FUNCTION

FUNCTION FC 200 : VOID
VERSION : 0.1
BEGIN
// (block stored without names or comments; labels and parameter names are numbered)
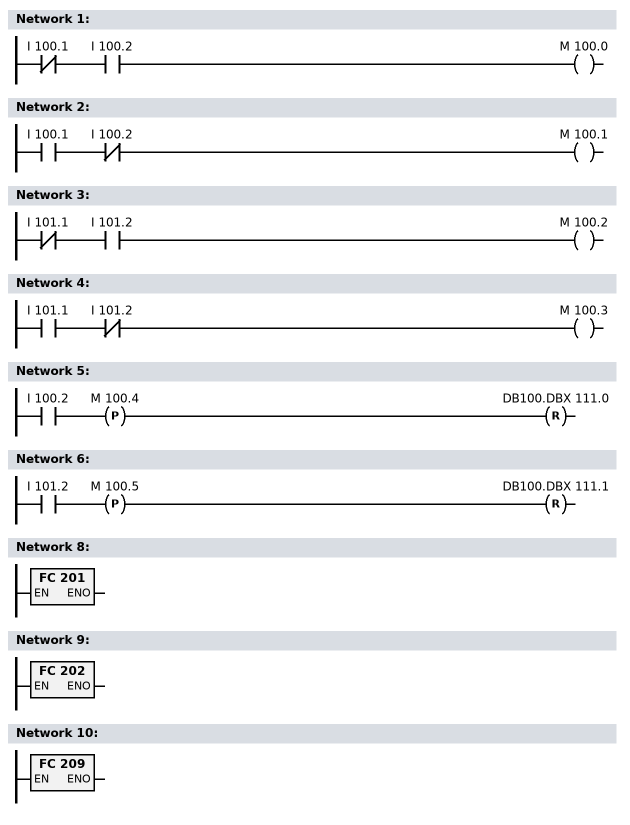
NETWORK
TITLE =
      AN    I 100.1;
      A     I 100.2;
      =     M 100.0;
NETWORK
TITLE =
      A     I 100.1;
      AN    I 100.2;
      =     M 100.1;
NETWORK
TITLE =
      AN    I 101.1;
      A     I 101.2;
      =     M 100.2;
NETWORK
TITLE =
      A     I 101.1;
      AN    I 101.2;
      =     M 100.3;
NETWORK
TITLE =
      A     I 100.2;
      FP    M 100.4;
      R     DB100.DBX 111.0;
NETWORK
TITLE =
      A     I 101.2;
      FP    M 100.5;
      R     DB100.DBX 111.1;
NETWORK
TITLE =
NETWORK
TITLE =
      CALL  FC 201;
      NOP   0;
NETWORK
TITLE =
      CALL  FC 202;
      NOP   0;
NETWORK
TITLE =
      CALL  FC 209;
      NOP   0;
END_FUNCTION

FUNCTION FC 201 : VOID
VERSION : 0.1
BEGIN
// (block stored without names or comments; labels and parameter names are numbered)
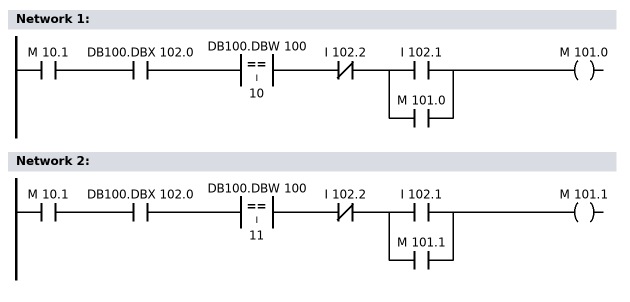
NETWORK
TITLE =
      A     M 10.1;
      A     DB100.DBX 102.0;
      A(;
      L     DB100.DBW 100;
      L     10;
      ==I;
      );
      AN    I 102.2;
      A(;
      O     I 102.1;
      O     M 101.0;
      );
      =     M 101.0;
NETWORK
TITLE =
      A     M 10.1;
      A     DB100.DBX 102.0;
      A(;
      L     DB100.DBW 100;
      L     11;
      ==I;
      );
      AN    I 102.2;
      A(;
      O     I 102.1;
      O     M 101.1;
      );
      =     M 101.1;
END_FUNCTION

FUNCTION FC 202 : VOID
VERSION : 0.1
BEGIN
// (block stored without names or comments; labels and parameter names are numbered)
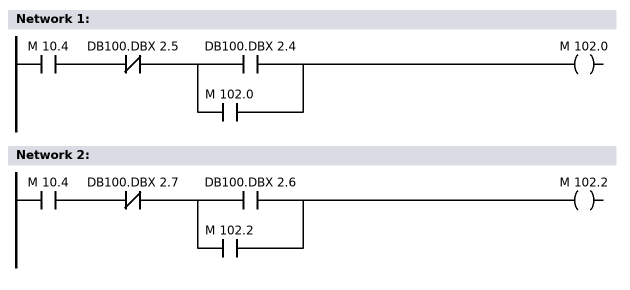
NETWORK
TITLE =
      A     M 10.4;
      AN    DB100.DBX 2.5;
      A(;
      O     DB100.DBX 2.4;
      O     M 102.0;
      );
      =     M 102.0;
NETWORK
TITLE =
      A     M 10.4;
      AN    DB100.DBX 2.7;
      A(;
      O     DB100.DBX 2.6;
      O     M 102.2;
      );
      =     M 102.2;
END_FUNCTION

FUNCTION FC 209 : VOID
VERSION : 0.1
BEGIN
// (block stored without names or comments; labels and parameter names are numbered)
